PROGRAM MAIN
VAR
END_VAR

P_Control();

END_PROGRAM

(* stored: Version 1.1.0.1, ProductVersion 3.1.4024.12
   POU MAIN: Id {86f126c1-91e1-4c3f-b185-3f74de79e12b}, SpecialFunc None *)
